FUNCTION_BLOCK FB_Motion2way
VAR_INPUT
	
	//advances
	iAdvanceAuto: BOOL; //auto request
	iAdvanceManual: BOOL; //manual request
	iAdvanceInterlock: BOOL; //must be TRUE to perform motion
	iAdvanceDepth: BOOL; //limit sensor for advanced
	iAdvancePrompt: BOOL; //TRUE if the motion is the next step in the sequence
	iAdvanceDelay:TIME := T#100MS; //advance delay

	iAdvanceTimeout:TIME := T#5S; //default timeout value
	
	//returns
	iReturnManual: BOOL; //manual request
	iReturnAuto: BOOL; //auto request
	iReturnInterlock: BOOL; //must be TRUE to perform motion
	iReturnTimeout:TIME := T#5S; //default timeout value
	iReturnDepth: BOOL; //limit sensor for advanced
	iReturnPrompt: BOOL; //TRUE if the motion is the next step in the sequence
	iReturnDelay:TIME := T#100MS; //return delay
	

	iLatchCoilOn: BOOL; //TRUE to latch the coil on after a motion
	

	
	iMode: typeStationMode; //what mode is station in?
	
	iRodlockTime:TIME:= T#250MS; //delay after rod lock release to perform motion
	iLatchOnRodLock:BOOL; //TRUE to latch on the rodlock on the motion (disables on loss of power)
	iDelayRodlockOff:BOOL; //TRUE to delay the rodlock signal off (sometimes prevent binding of 
	iUseRodlockDelay:BOOL; //TRUE to delay the valve cylinder untill the rodlock has been fired, for a time
	iCheckSwitchFaultsOff:BOOL :=FALSE; //TRUE to check if switch faults for double off conditions
	iLatchOnLimitSwitch:BOOL:=TRUE; //TRUE to latch the output on the limit switch (normal cylinder)
	iEnergiseOnPowerOn:BOOL:=TRUE; //TRUE to apply coil when powered on if limit switch is TRUE
	iIgnoreLostSwitchFault:BOOL:=FALSE; //TRUE to ignore lost switch fault states (some use cases)



END_VAR
VAR_OUTPUT

	//advance coil
	qAdvanceCoil: BOOL;
	qAdvancedDepth: BOOL;
	qAdvanceTime: TIME;
	qAdvancePrompt: BOOL;
	qAdvanceInterlock: BOOL;

	
	//return coil
	qReturnCoil: BOOL;
	qReturnDepth: BOOL;
	qReturnTime: TIME;
	qReturnPrompt: BOOL;
	qReturnInterlock: BOOL;

	
	qFaultAdvanceTimeout: BOOL;		//TRUE if the advance switch was not reached
	qFaultReturnTimeout: BOOL;		//TRUE if the return switch was not reached
	qFaultLostAdvance: BOOL;		//TRUE if the advance switch was lost after advancing
	qFaultLostReturn: BOOL;			//TRUE if the return switch was lost after advancing
	qSwitchFault: BOOL;				//TRUE if Both the advance and return switch were TRUE

	

	qRodLock: BOOL; //connect to rodlock valve
END_VAR
VAR
	
	//advance variables
	tAdvanceReq: BOOL;
	timAdvanceTimer: TON;
	tAdvanceTimeoutFault: BOOL;
	tAdvanceWithInterlock: BOOL;
	
	//return variables
	tReturnReq: BOOL;
	timReturnTimer: TON;
	tReturnTimeoutFault: BOOL;
	tReturnWithInterlock: BOOL;
	
	
	timSwitchFault: TON;
	
	timRodLockRelease: TON;
	// Energise rodlock or raillock
	tEnableRodlock: BOOL;
	
	
	tRodlockSignal: BOOL;
	timRodlockOffDelay: TOF;
	timAdvanceDelay: TON;
	tAdvanced: BOOL;
	timReturnDelay: TON;
	tReturned: BOOL;
	timAdvanceDelayOff: TOF;
	timReturnDelayOff: tof;
	
	osrAdvancePowerOn: R_TRIG;
	osrReturnPowerOn: R_TRIG;
END_VAR
VAR // added by the converter: edge detectors and wires of the graphical bodies
    _ft1, _ft2, _ft3, _ft4, _ft5, _ft6, _ft7 : F_TRIG;
    _w1, _w2 : BOOL;
END_VAR

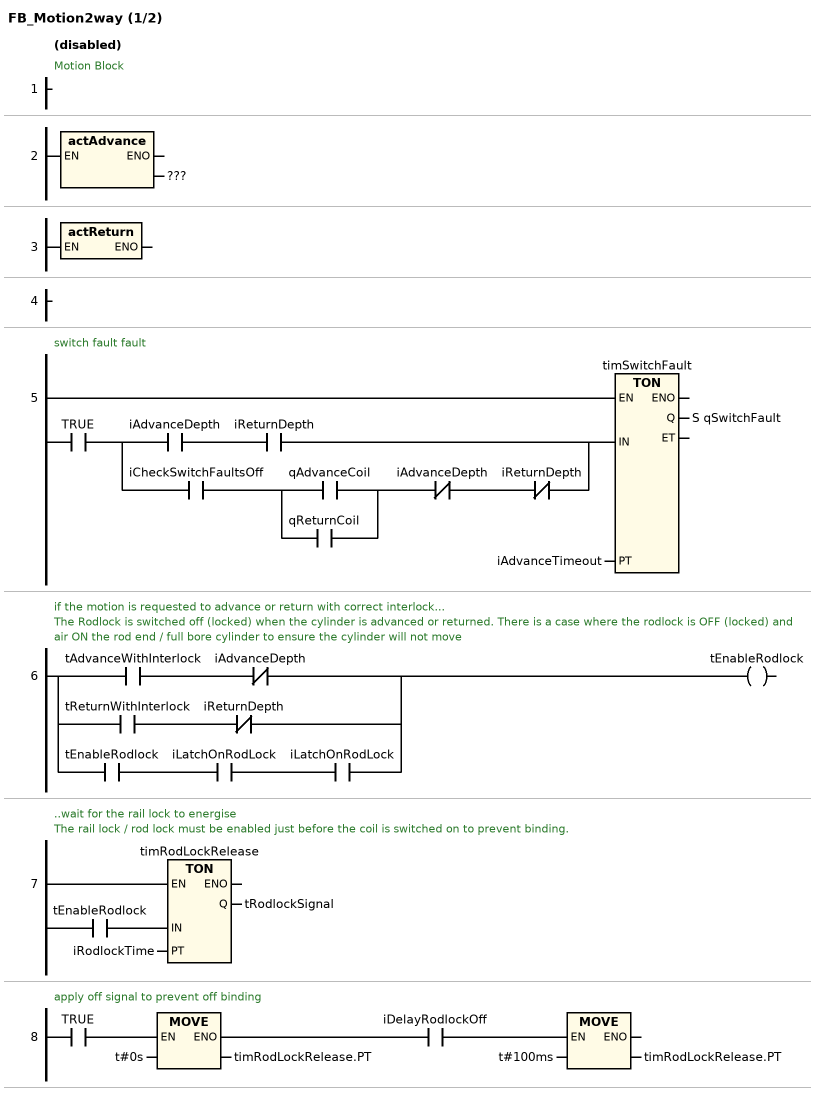
// NETWORK 1 (disabled)
// Motion Block

// NETWORK 2
actAdvance();

// NETWORK 3
actReturn();

// NETWORK 4

// NETWORK 5
// switch fault fault
timSwitchFault(IN := TRUE AND (iAdvanceDepth AND iReturnDepth OR iCheckSwitchFaultsOff AND (qAdvanceCoil OR qReturnCoil) AND NOT iAdvanceDepth AND NOT iReturnDepth), PT := iAdvanceTimeout); // TON
qSwitchFault S= timSwitchFault.Q;

// NETWORK 6
// if the motion is requested to advance or return with correct interlock...
// The Rodlock is switched off (locked) when the cylinder is advanced or returned. There is a case where the rodlock is OFF (locked) and air ON the rod end / full bore cylinder to ensure the cylinder will not move
tEnableRodlock := tAdvanceWithInterlock AND NOT iAdvanceDepth OR tReturnWithInterlock AND NOT iReturnDepth OR tEnableRodlock AND iLatchOnRodLock AND iLatchOnRodLock;

// NETWORK 7
// ..wait for the rail lock to energise
// The rail lock / rod lock must be enabled just before the coil is switched on to prevent binding.
timRodLockRelease(IN := tEnableRodlock, PT := iRodlockTime, Q => tRodlockSignal); // TON

// NETWORK 8
// apply off signal to prevent off binding
timRodLockRelease.PT := t#0s;
IF TRUE AND iDelayRodlockOff THEN timRodLockRelease.PT := t#100ms; END_IF

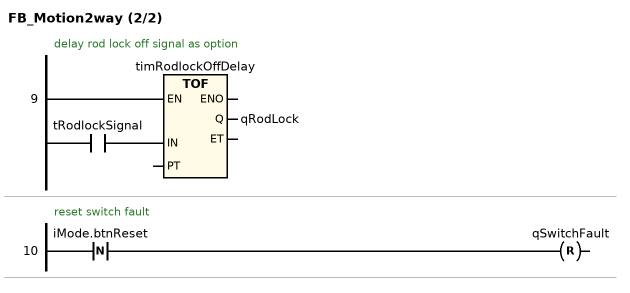
// NETWORK 9
// delay rod lock off signal as option
timRodlockOffDelay(IN := tRodlockSignal, Q => qRodLock); // TOF

// NETWORK 10
// reset switch fault
_ft1(CLK := iMode.btnReset);
qSwitchFault R= _ft1.Q;

ACTION actAdvance:
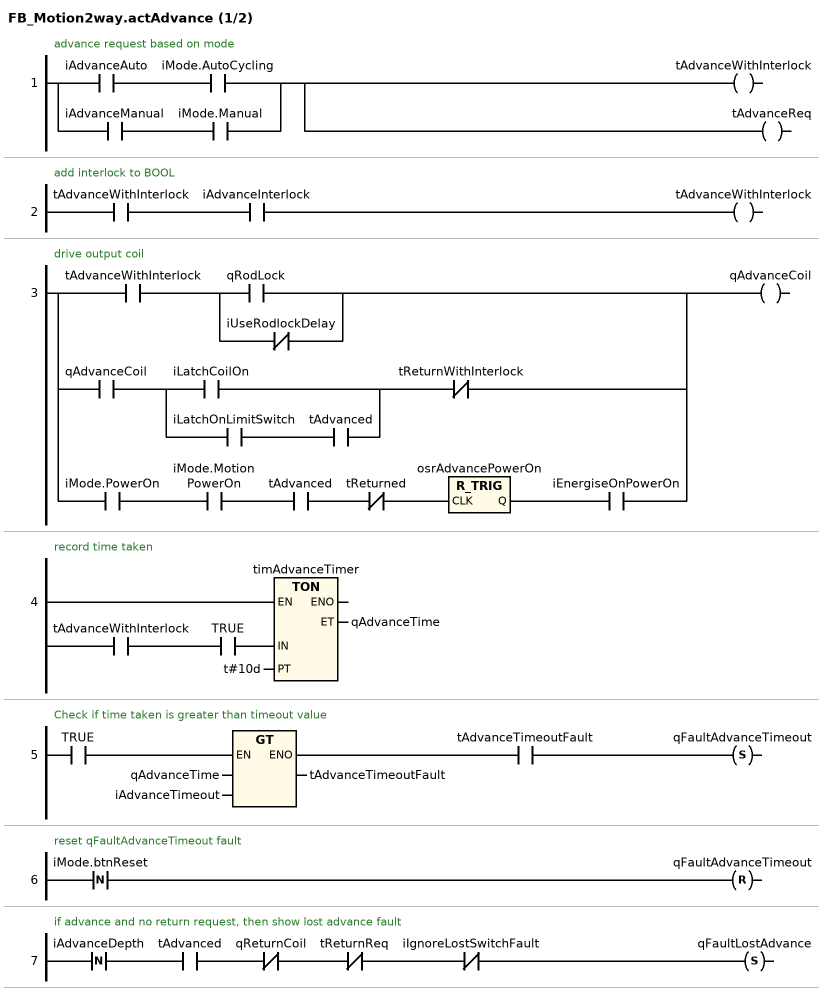
// NETWORK 1
// advance request based on mode
_w1 := iAdvanceAuto AND iMode.AutoCycling OR iAdvanceManual AND iMode.Manual;
tAdvanceWithInterlock := _w1;
tAdvanceReq := _w1;

// NETWORK 2
// add interlock to BOOL
tAdvanceWithInterlock := tAdvanceWithInterlock AND iAdvanceInterlock;

// NETWORK 3
// drive output coil
osrAdvancePowerOn(CLK := iMode.PowerOn AND iMode.MotionPowerOn AND tAdvanced AND NOT tReturned); // R_TRIG
qAdvanceCoil := tAdvanceWithInterlock AND (qRodLock OR NOT iUseRodlockDelay) OR qAdvanceCoil AND (iLatchCoilOn OR iLatchOnLimitSwitch AND tAdvanced) AND NOT tReturnWithInterlock OR osrAdvancePowerOn.Q AND iEnergiseOnPowerOn;

// NETWORK 4
// record time taken
timAdvanceTimer(IN := tAdvanceWithInterlock AND TRUE, PT := t#10d, ET => qAdvanceTime); // TON

// NETWORK 5
// Check if time taken is greater than timeout value
tAdvanceTimeoutFault := qAdvanceTime > iAdvanceTimeout;
qFaultAdvanceTimeout S= TRUE AND tAdvanceTimeoutFault;

// NETWORK 6
// reset qFaultAdvanceTimeout fault
_ft2(CLK := iMode.btnReset);
qFaultAdvanceTimeout R= _ft2.Q;

// NETWORK 7
// if advance and no return request, then show lost advance fault
_ft3(CLK := iAdvanceDepth);
qFaultLostAdvance S= _ft3.Q AND tAdvanced AND NOT qReturnCoil AND NOT tReturnReq AND NOT iIgnoreLostSwitchFault;

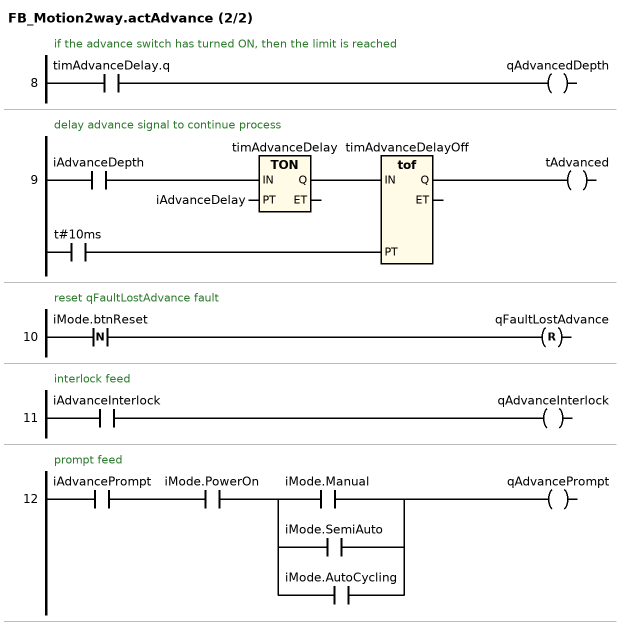
// NETWORK 8
// if the advance switch has turned ON, then the limit is reached
qAdvancedDepth := timAdvanceDelay.q;

// NETWORK 9
// delay advance signal to continue process
timAdvanceDelay(IN := iAdvanceDepth, PT := iAdvanceDelay); // TON
timAdvanceDelayOff(IN := timAdvanceDelay.Q, PT := t#10ms); // tof
tAdvanced := timAdvanceDelayOff.Q;

// NETWORK 10
// reset qFaultLostAdvance fault
_ft4(CLK := iMode.btnReset);
qFaultLostAdvance R= _ft4.Q;

// NETWORK 11
// interlock feed
qAdvanceInterlock := iAdvanceInterlock;

// NETWORK 12
// prompt feed
qAdvancePrompt := iAdvancePrompt AND iMode.PowerOn AND (iMode.Manual OR iMode.SemiAuto OR iMode.AutoCycling);
END_ACTION

ACTION actReturn:
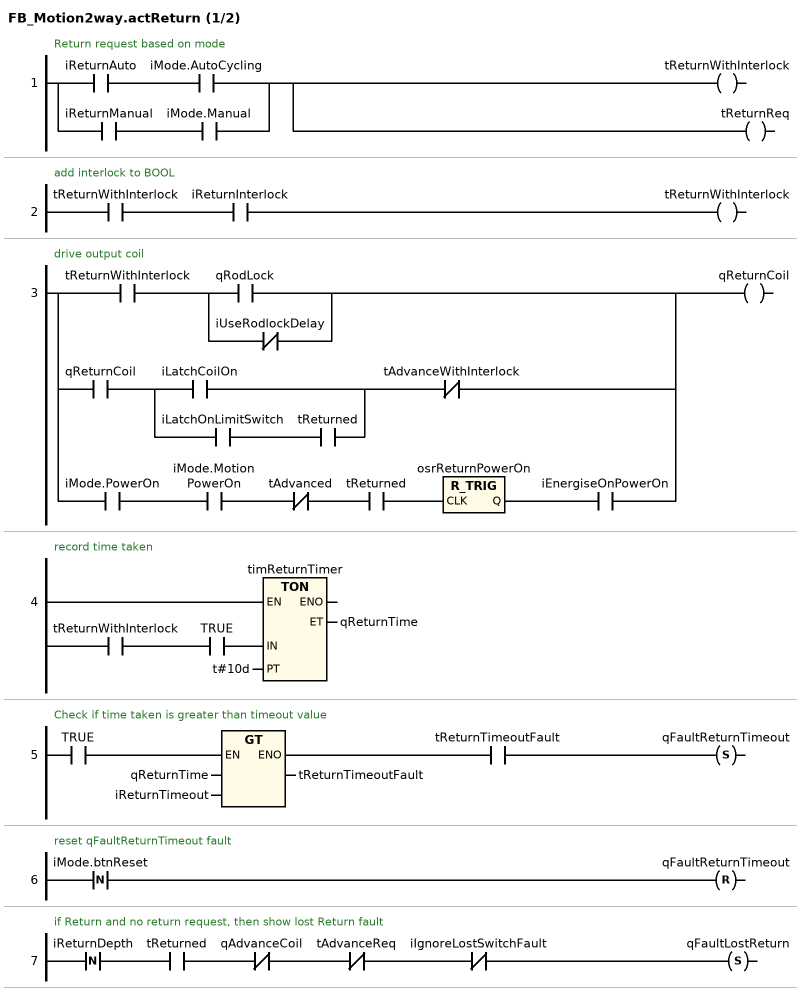
// NETWORK 1
// Return request based on mode
_w2 := iReturnAuto AND iMode.AutoCycling OR iReturnManual AND iMode.Manual;
tReturnWithInterlock := _w2;
tReturnReq := _w2;

// NETWORK 2
// add interlock to BOOL
tReturnWithInterlock := tReturnWithInterlock AND iReturnInterlock;

// NETWORK 3
// drive output coil
osrReturnPowerOn(CLK := iMode.PowerOn AND iMode.MotionPowerOn AND NOT tAdvanced AND tReturned); // R_TRIG
qReturnCoil := tReturnWithInterlock AND (qRodLock OR NOT iUseRodlockDelay) OR qReturnCoil AND (iLatchCoilOn OR iLatchOnLimitSwitch AND tReturned) AND NOT tAdvanceWithInterlock OR osrReturnPowerOn.Q AND iEnergiseOnPowerOn;

// NETWORK 4
// record time taken
timReturnTimer(IN := tReturnWithInterlock AND TRUE, PT := t#10d, ET => qReturnTime); // TON

// NETWORK 5
// Check if time taken is greater than timeout value
tReturnTimeoutFault := qReturnTime > iReturnTimeout;
qFaultReturnTimeout S= TRUE AND tReturnTimeoutFault;

// NETWORK 6
// reset qFaultReturnTimeout fault
_ft5(CLK := iMode.btnReset);
qFaultReturnTimeout R= _ft5.Q;

// NETWORK 7
// if Return and no return request, then show lost Return fault
_ft6(CLK := iReturnDepth);
qFaultLostReturn S= _ft6.Q AND tReturned AND NOT qAdvanceCoil AND NOT tAdvanceReq AND NOT iIgnoreLostSwitchFault;

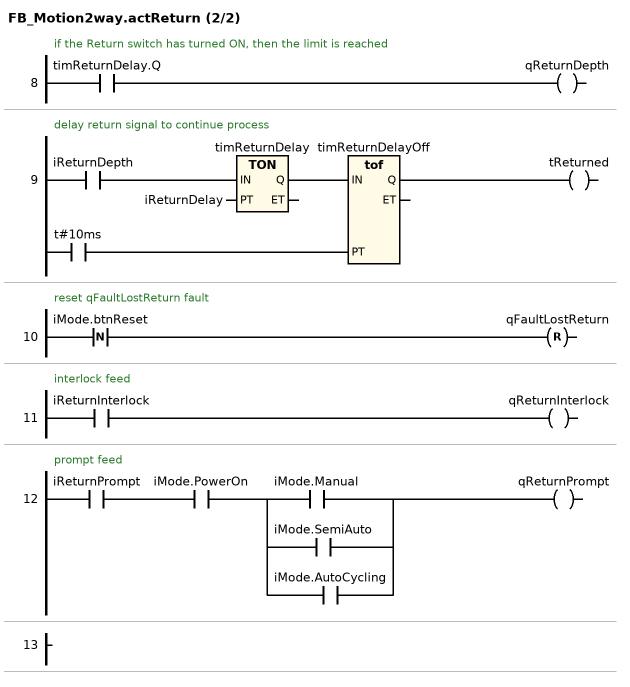
// NETWORK 8
// if the Return switch has turned ON, then the limit is reached
qReturnDepth := timReturnDelay.Q;

// NETWORK 9
// delay return signal to continue process
timReturnDelay(IN := iReturnDepth, PT := iReturnDelay); // TON
timReturnDelayOff(IN := timReturnDelay.Q, PT := t#10ms); // tof
tReturned := timReturnDelayOff.Q;

// NETWORK 10
// reset qFaultLostReturn fault
_ft7(CLK := iMode.btnReset);
qFaultLostReturn R= _ft7.Q;

// NETWORK 11
// interlock feed
qReturnInterlock := iReturnInterlock;

// NETWORK 12
// prompt feed
qReturnPrompt := iReturnPrompt AND iMode.PowerOn AND (iMode.Manual OR iMode.SemiAuto OR iMode.AutoCycling);

// NETWORK 13
END_ACTION

END_FUNCTION_BLOCK

(* stored: Version 1.1.0.1, ProductVersion 3.1.4024.11
   POU FB_Motion2way: Id {67c13904-6fb4-438d-a287-3bdbf007bb70}, SpecialFunc None
   Action actAdvance: Id {24e21505-d2b3-4004-8ac5-a7f8d2c0aa31}
   Action actReturn: Id {fb3fca72-cf67-4645-8604-ff2fefc5f3e0} *)
